# B&R Automation Studio project ControllerSim
Automation Studio 4.12.2.93

## Configuration Simulation

### Hardware
```
5APC2200_AL14_000 : 5APC2200.AL14-000 v2.0.7.0
  Connector IF3:
    AssignedOperatingSystem = ARemb
    ActivateDevice = 1
  Connector IF4:
    AssignedOperatingSystem = ARemb
    ActivateDevice = 1
  Connector IF5:
    AssignedOperatingSystem = ARemb
  Connector IF6:
    AssignedOperatingSystem = ARemb
  ConfigurationID = ControllerSim_Simulation
  Simulation = 1
```

## Logical view

### Global.var
```iecst
VAR
	gCounter : USINT;
	flag : BOOL := TRUE;
END_VAR
```

### Program Logical/Program

#### Main.st
```iecst
PROGRAM _INIT
	(* Insert code here *)
	gCounter:=0;
	 flag :=TRUE;
END_PROGRAM

PROGRAM _CYCLIC
	IF flag = TRUE THEN
		gCounter := gCounter + 1;
	END_IF

END_PROGRAM

PROGRAM _EXIT
	(* Insert code here *)

END_PROGRAM
```
